FUNCTION_BLOCK CROSS_JOYSTICK (* Behaves like a cross-joystick: transitions between directional states (LEFT, RIGHT, UP, DOWN) must go through CENTER. *)
  (* Standard: 61499-2; Description: Copyright (c) 2026 HR Agrartechnik GmbH *)
  (* Version 1.0, 2026-06-11, Franz Höpfinger, HR Agrartechnik GmbH, Initial implementation of Cross-Joystick *)
  PACKAGE logiBUS::signalprocessing::interlock;
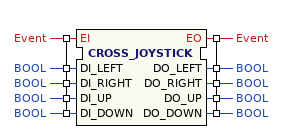
  EVENT_INPUT
    EI WITH DI_LEFT, DI_RIGHT, DI_UP, DI_DOWN;
  END_EVENT
  EVENT_OUTPUT
    EO WITH DO_LEFT, DO_RIGHT, DO_UP, DO_DOWN;
  END_EVENT
  VAR_INPUT
    DI_LEFT : BOOL; (* Joystick Left position switch *)
    DI_RIGHT : BOOL; (* Joystick Right position switch *)
    DI_UP : BOOL; (* Joystick Up position switch *)
    DI_DOWN : BOOL; (* Joystick Down position switch *)
  END_VAR
  VAR_OUTPUT
    DO_LEFT : BOOL; (* Output Left indicator *)
    DO_RIGHT : BOOL; (* Output Right indicator *)
    DO_UP : BOOL; (* Output Up indicator *)
    DO_DOWN : BOOL; (* Output Down indicator *)
  END_VAR
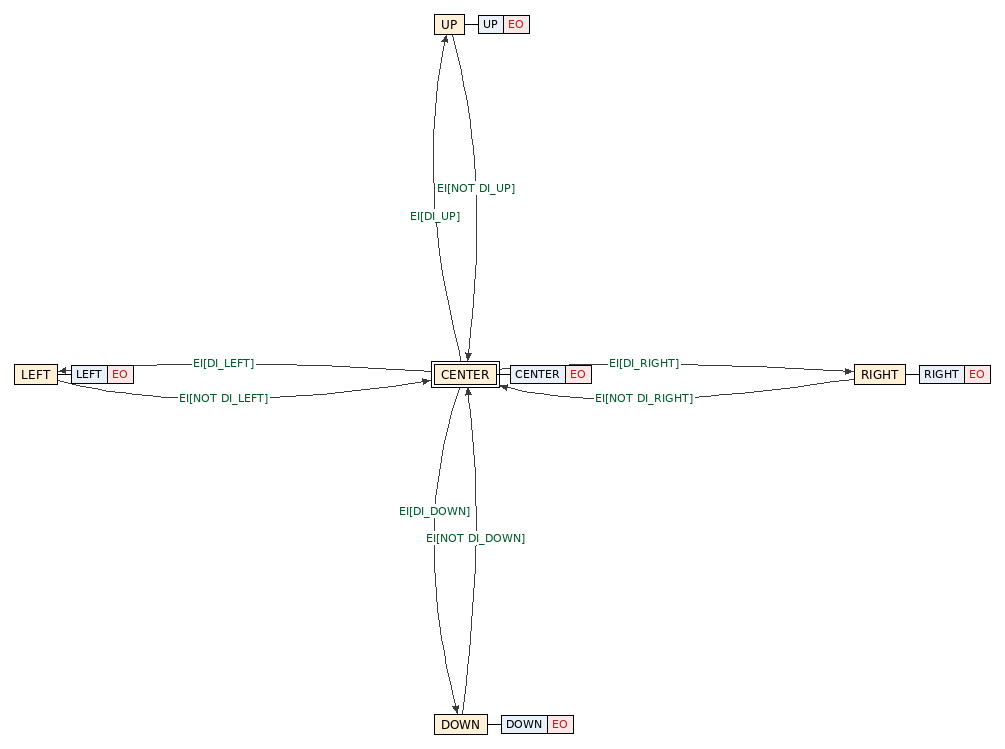
  EC_STATES
    CENTER : CENTER -> EO;
    LEFT : LEFT -> EO;
    RIGHT : RIGHT -> EO;
    UP : UP -> EO;
    DOWN : DOWN -> EO;
  END_STATES
  EC_TRANSITIONS
    CENTER TO LEFT := EI[DI_LEFT];
    CENTER TO RIGHT := EI[DI_RIGHT];
    CENTER TO UP := EI[DI_UP];
    CENTER TO DOWN := EI[DI_DOWN];
    LEFT TO CENTER := EI[NOT DI_LEFT];
    RIGHT TO CENTER := EI[NOT DI_RIGHT];
    UP TO CENTER := EI[NOT DI_UP];
    DOWN TO CENTER := EI[NOT DI_DOWN];
  END_TRANSITIONS
  ALGORITHM CENTER IN ST:
DO_LEFT := BOOL#FALSE;
DO_RIGHT := BOOL#FALSE;
DO_UP := BOOL#FALSE;
DO_DOWN := BOOL#FALSE;
  END_ALGORITHM
  ALGORITHM LEFT IN ST:
DO_LEFT := BOOL#TRUE;
DO_RIGHT := BOOL#FALSE;
DO_UP := BOOL#FALSE;
DO_DOWN := BOOL#FALSE;
  END_ALGORITHM
  ALGORITHM RIGHT IN ST:
DO_LEFT := BOOL#FALSE;
DO_RIGHT := BOOL#TRUE;
DO_UP := BOOL#FALSE;
DO_DOWN := BOOL#FALSE;
  END_ALGORITHM
  ALGORITHM UP IN ST:
DO_LEFT := BOOL#FALSE;
DO_RIGHT := BOOL#FALSE;
DO_UP := BOOL#TRUE;
DO_DOWN := BOOL#FALSE;
  END_ALGORITHM
  ALGORITHM DOWN IN ST:
DO_LEFT := BOOL#FALSE;
DO_RIGHT := BOOL#FALSE;
DO_UP := BOOL#FALSE;
DO_DOWN := BOOL#TRUE;
  END_ALGORITHM
END_FUNCTION_BLOCK
